// TIA Portal V17 export
// export: Created 2025-06-26T06:49:29.000062Z, ExportSetting WithDefaults, DisplayName Totally Integrated Automation Portal, DisplayVersion V17 Update 8, DisplayName TIA Portal Openness, DisplayVersion V17 Update 8, DisplayName TIA Portal Version Control Interface, DisplayVersion V17, DisplayName STEP 7 Professional, DisplayVersion V17 Update 8, DisplayName STEP 7 Safety, DisplayVersion V17 Update 6, DisplayName WinCC Advanced, DisplayVersion V17 Update 8
TYPE "stET200AL_DIQ_I"
// stored: IsFailsafeCompliant false
   STRUCT
      DI00 : Bool;
      DI01 : Bool;
      DI02 : Bool;
      DI03 : Bool;
      DI04 : Bool;
      DI05 : Bool;
      DI06 : Bool;
      DI07 : Bool;
      DI08 : Bool;
      DI09 : Bool;
      DI10 : Bool;
      DI11 : Bool;
      DI12 : Bool;
      DI13 : Bool;
      DI14 : Bool;
      DI15 : Bool;
      STAT : Array[0..31] of Bool;   // "Value Status" checked in module parameters
   END_STRUCT;
END_TYPE
